PROGRAM TowerLightCtrl
VAR
	TLctrl					: fbTowerLightCtrl;
	CLKPLS					: CLOCK_PLS;
	CP						: BOOL;
	SFQ						: BOOL;

	ARbAlarmOutput421RE		: R_TRIG;
	ARbAlarmOutput422RE		: R_TRIG;
	ARbAlarmOutput424RE		: R_TRIG;
	ARbAlarmOutput425RE		: R_TRIG;
	ARbAlarmOutput113RE		: R_TRIG;

	ARbAlarmOutput423RE		: R_TRIG;
	ARbAlarmOutput426RE		: R_TRIG;
	ARbAlarmOutput429RE		: R_TRIG;

	bAlarmOccurFlagIND		: BOOL;
	bBuzzerFlagIND			: BOOL;

END_VAR
VAR // added by the converter: edge detectors and wires of the graphical bodies
    _w1 : BOOL;
END_VAR

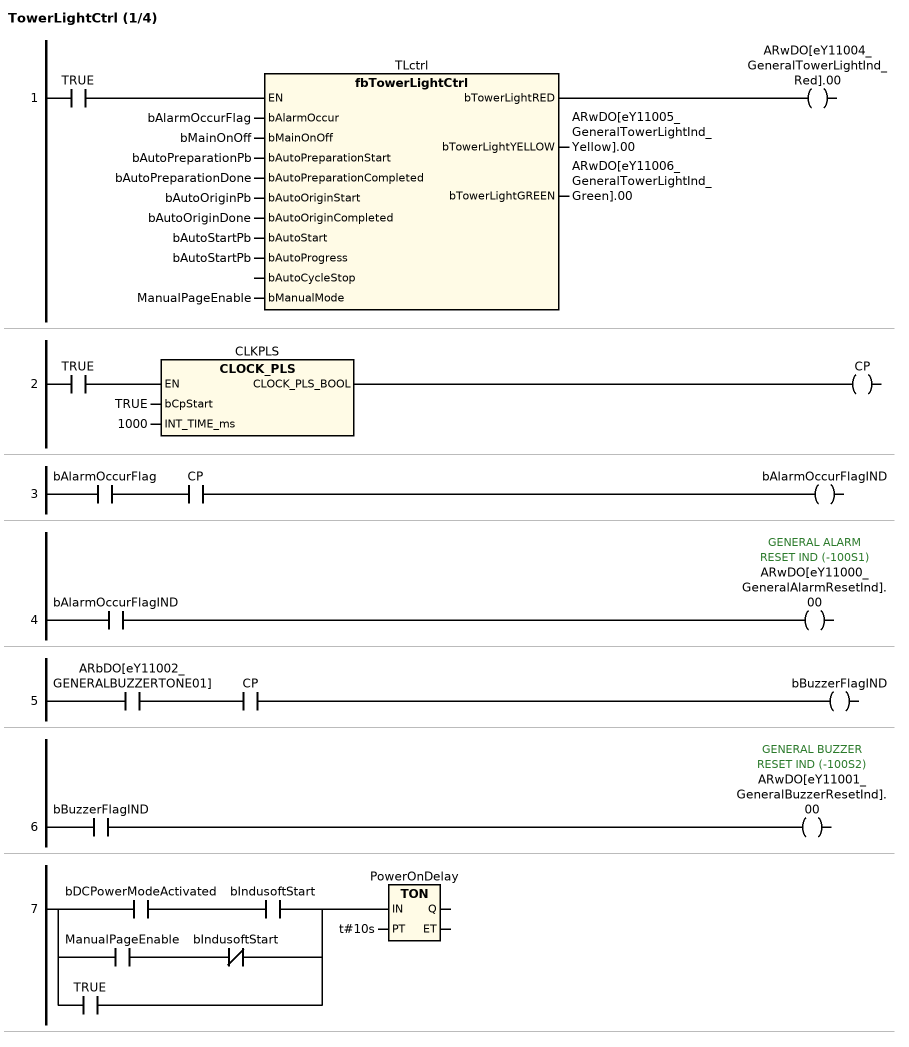
// NETWORK 1
TLctrl(
    bAlarmOccur := bAlarmOccurFlag,
    bMainOnOff := bMainOnOff,
    bAutoPreparationStart := bAutoPreparationPb,
    bAutoPreparationCompleted := bAutoPreparationDone,
    bAutoOriginStart := bAutoOriginPb,
    bAutoOriginCompleted := bAutoOriginDone,
    bAutoStart := bAutoStartPb,
    bAutoProgress := bAutoStartPb,
    bManualMode := ManualPageEnable,
    bTowerLightYELLOW => ARwDO[eY11005_GeneralTowerLightInd_Yellow].00,
    bTowerLightGREEN => ARwDO[eY11006_GeneralTowerLightInd_Green].00); // fbTowerLightCtrl
ARwDO[eY11004_GeneralTowerLightInd_Red].00 := TLctrl.bTowerLightRED;

// NETWORK 2
CLKPLS(bCpStart := TRUE, INT_TIME_ms := 1000); // CLOCK_PLS
CP := CLKPLS.CLOCK_PLS_BOOL;

// NETWORK 3
bAlarmOccurFlagIND := bAlarmOccurFlag AND CP;

// NETWORK 4
//   ARwDO[eY11000_GeneralAlarmResetInd].00: GENERAL ALARM RESET IND (-100S1)
ARwDO[eY11000_GeneralAlarmResetInd].00 := bAlarmOccurFlagIND;

// NETWORK 5
bBuzzerFlagIND := ARbDO[eY11002_GENERALBUZZERTONE01] AND CP;

// NETWORK 6
//   ARwDO[eY11001_GeneralBuzzerResetInd].00: GENERAL BUZZER RESET IND (-100S2)
ARwDO[eY11001_GeneralBuzzerResetInd].00 := bBuzzerFlagIND;

// NETWORK 7
PowerOnDelay(IN := bDCPowerModeActivated AND bIndusoftStart OR ManualPageEnable AND NOT bIndusoftStart OR TRUE, PT := t#10s); // TON

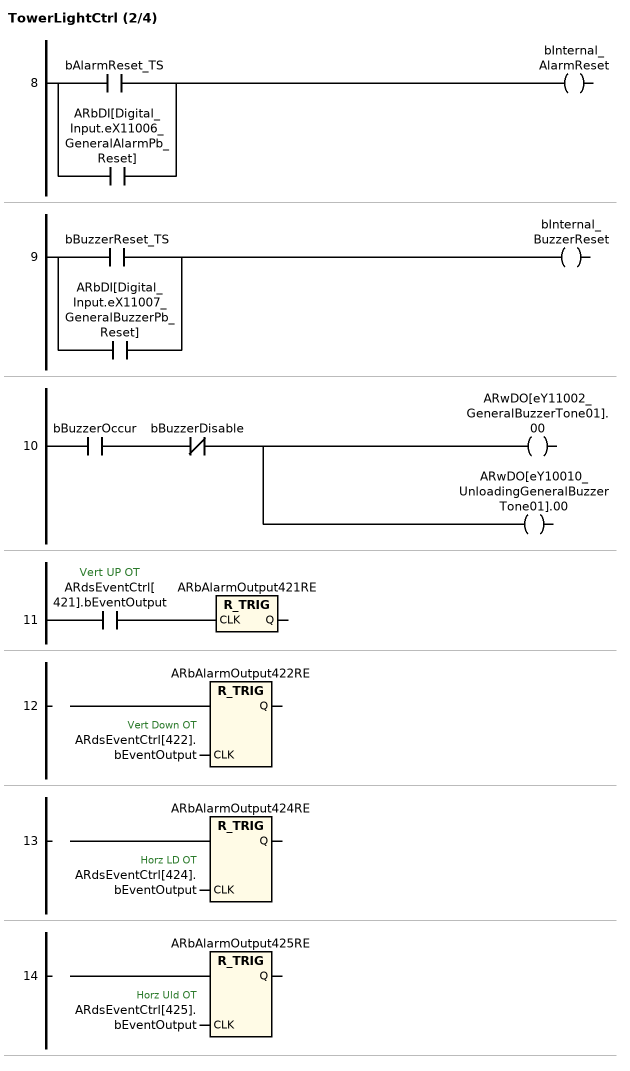
// NETWORK 8
bInternal_AlarmReset := bAlarmReset_TS OR ARbDI[Digital_Input.eX11006_GeneralAlarmPb_Reset];

// NETWORK 9
bInternal_BuzzerReset := bBuzzerReset_TS OR ARbDI[Digital_Input.eX11007_GeneralBuzzerPb_Reset];

// NETWORK 10
_w1 := bBuzzerOccur AND NOT bBuzzerDisable;
ARwDO[eY11002_GeneralBuzzerTone01].00 := _w1;
ARwDO[eY10010_UnloadingGeneralBuzzerTone01].00 := _w1;

// NETWORK 11
//   ARdsEventCtrl[421].bEventOutput: Vert UP OT
ARbAlarmOutput421RE(CLK := ARdsEventCtrl[421].bEventOutput); // R_TRIG

// NETWORK 12
//   ARdsEventCtrl[422].bEventOutput: Vert Down OT
ARbAlarmOutput422RE(CLK := ARdsEventCtrl[422].bEventOutput); // R_TRIG

// NETWORK 13
//   ARdsEventCtrl[424].bEventOutput: Horz LD OT
ARbAlarmOutput424RE(CLK := ARdsEventCtrl[424].bEventOutput); // R_TRIG

// NETWORK 14
//   ARdsEventCtrl[425].bEventOutput: Horz Uld OT
ARbAlarmOutput425RE(CLK := ARdsEventCtrl[425].bEventOutput); // R_TRIG

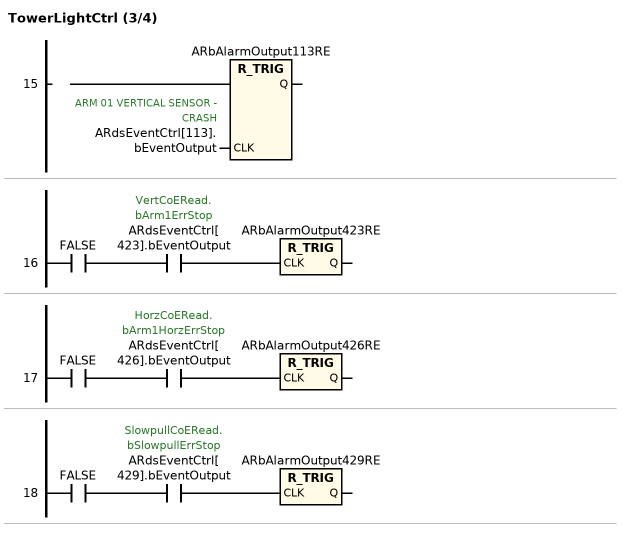
// NETWORK 15
//   ARdsEventCtrl[113].bEventOutput: ARM 01 VERTICAL SENSOR - CRASH
ARbAlarmOutput113RE(CLK := ARdsEventCtrl[113].bEventOutput); // R_TRIG

// NETWORK 16
//   ARdsEventCtrl[423].bEventOutput: VertCoERead.bArm1ErrStop
ARbAlarmOutput423RE(CLK := FALSE AND ARdsEventCtrl[423].bEventOutput); // R_TRIG

// NETWORK 17
//   ARdsEventCtrl[426].bEventOutput: HorzCoERead.bArm1HorzErrStop
ARbAlarmOutput426RE(CLK := FALSE AND ARdsEventCtrl[426].bEventOutput); // R_TRIG

// NETWORK 18
//   ARdsEventCtrl[429].bEventOutput: SlowpullCoERead.bSlowpullErrStop
ARbAlarmOutput429RE(CLK := FALSE AND ARdsEventCtrl[429].bEventOutput); // R_TRIG

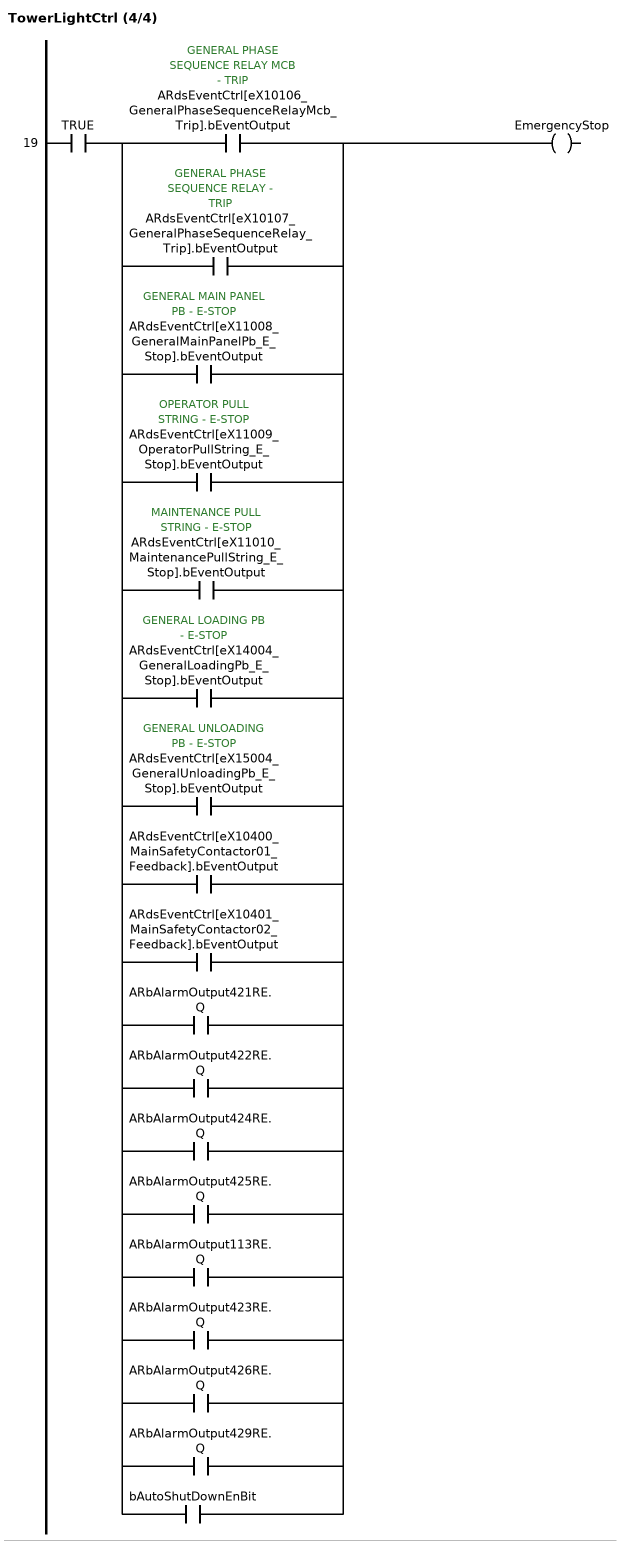
// NETWORK 19
//   ARdsEventCtrl[eX10106_GeneralPhaseSequenceRelayMcb_Trip].bEventOutput: GENERAL PHASE SEQUENCE RELAY MCB - TRIP
//   ARdsEventCtrl[eX10107_GeneralPhaseSequenceRelay_Trip].bEventOutput: GENERAL PHASE SEQUENCE RELAY - TRIP
//   ARdsEventCtrl[eX11008_GeneralMainPanelPb_E_Stop].bEventOutput: GENERAL MAIN PANEL PB - E-STOP
//   ARdsEventCtrl[eX11009_OperatorPullString_E_Stop].bEventOutput: OPERATOR PULL STRING - E-STOP
//   ARdsEventCtrl[eX11010_MaintenancePullString_E_Stop].bEventOutput: MAINTENANCE PULL STRING - E-STOP
//   ARdsEventCtrl[eX14004_GeneralLoadingPb_E_Stop].bEventOutput: GENERAL LOADING PB - E-STOP
//   ARdsEventCtrl[eX15004_GeneralUnloadingPb_E_Stop].bEventOutput: GENERAL UNLOADING PB - E-STOP
EmergencyStop := TRUE AND (ARdsEventCtrl[eX10106_GeneralPhaseSequenceRelayMcb_Trip].bEventOutput OR ARdsEventCtrl[eX10107_GeneralPhaseSequenceRelay_Trip].bEventOutput OR ARdsEventCtrl[eX11008_GeneralMainPanelPb_E_Stop].bEventOutput OR ARdsEventCtrl[eX11009_OperatorPullString_E_Stop].bEventOutput OR ARdsEventCtrl[eX11010_MaintenancePullString_E_Stop].bEventOutput OR ARdsEventCtrl[eX14004_GeneralLoadingPb_E_Stop].bEventOutput OR ARdsEventCtrl[eX15004_GeneralUnloadingPb_E_Stop].bEventOutput OR ARdsEventCtrl[eX10400_MainSafetyContactor01_Feedback].bEventOutput OR ARdsEventCtrl[eX10401_MainSafetyContactor02_Feedback].bEventOutput OR ARbAlarmOutput421RE.Q OR ARbAlarmOutput422RE.Q OR ARbAlarmOutput424RE.Q OR ARbAlarmOutput425RE.Q OR ARbAlarmOutput113RE.Q OR ARbAlarmOutput423RE.Q OR ARbAlarmOutput426RE.Q OR ARbAlarmOutput429RE.Q OR bAutoShutDownEnBit);

END_PROGRAM

(* stored: Version 1.1.0.1, ProductVersion 3.1.4024.12
   POU TowerLightCtrl: Id {b10ad78a-0a7b-4376-9e8a-73ab50aea843}, SpecialFunc None *)
